FUNCTION Convert_BYTE_TO_DT : BOOL
VAR_INPUT
	in : BYTE;
	out : REFERENCE TO DT;
END_VAR
VAR
	converted : DT;
END_VAR

converted := BYTE_TO_DT(in);

IF (DT_TO_BYTE(converted) <> in) THEN
	RETURN;
END_IF

out := converted;
Convert_BYTE_TO_DT := TRUE;

END_FUNCTION

(* stored: Version 1.1.0.1, ProductVersion 3.1.4024.12
   POU Convert_BYTE_TO_DT: Id {b7a25f8f-ae31-473f-93cf-37e960625455}, SpecialFunc None *)
